(*
	Custom MEMCPY function with a swap flag. 
	If bSwap is true and the length is within the range of 0 to 8, the memcpy operation will be performed with reversed byte order.
*) 
FUNCTION F_Memcpy : UDINT
VAR_INPUT
	destAddr 	: PVOID; //Destination Addr
	srcAddr 	: PVOID; //Source Addr
	n			: UDINT; //Bytes Length
	bSwap		: BOOL; //If TRUE and the length is within the range of 0 to 8, the memcpy operation will be performed with reversed byte order
END_VAR

VAR
	i 			: UDINT;
	aBuffer 	: ARRAY [0..7] OF BYTE;
	nWWORD		: WORD;
	nDWORD		: DWORD;
	nLWORD		: LWORD;
END_VAR

IF NOT bSWAP OR n > 8 THEN
	F_MEMCPY := MEMCPY(destAddr, srcAddr, n);
	RETURN;
END_IF

F_MEMCPY := MEMCPY(ADR(aBuffer), srcAddr, n);

FOR i:= 1 TO n DO	
	MEMCPY(destAddr + i - 1, ADR(aBuffer) + n - i, 1);
END_FOR

END_FUNCTION

(* stored: Version 1.1.0.1, ProductVersion 3.1.4024.12
   POU F_Memcpy: Id {4e35e276-b813-0523-07d7-44894b6f8e68}, SpecialFunc None *)
